(* PLC project Sem nome, Desconhecido Sem nome 1 *)
(* stored: creationDateTime 2019-12-04T19:50:12, modificationDateTime 2019-12-09T14:24:14 *)

PROGRAM Teste1
  VAR
    LIGA_PID AT %QX0.0 : BOOL;
    AUTO_PID AT %QX0.1 : BOOL;
  END_VAR
  VAR RETAIN
    SP AT %MD0 : REAL;
  END_VAR
  VAR
    VP AT %MD1 : REAL;
    SC AT %MD2 : REAL;
  END_VAR
  VAR RETAIN
    KP AT %MD3 : REAL;
    TI AT %MD4 : REAL;
    TD AT %MD5 : REAL;
  END_VAR
  VAR
    VP_RAW AT %IW100 : UINT;
    SC_RAW AT %QW101 : UINT;
  END_VAR
  VAR
    PID0 : PID;
  END_VAR

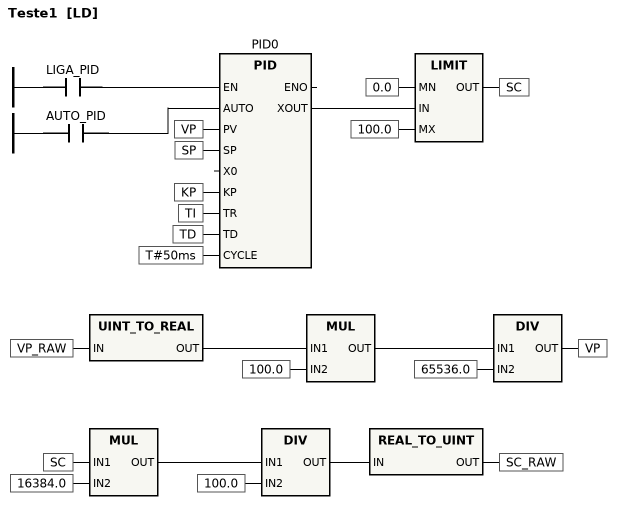
(* LD diagram, written out as Structured Text *)
VP := UINT_TO_REAL(VP_RAW) * 100.0 / 65536.0;
PID0(EN := LIGA_PID, AUTO := AUTO_PID, PV := VP, SP := SP, KP := KP, TR := TI, TD := TD, CYCLE := T#50ms);
SC := LIMIT(0.0, PID0.XOUT, 100.0);
SC_RAW := REAL_TO_UINT(SC * 16384.0 / 100.0);
END_PROGRAM

CONFIGURATION Config0
  RESOURCE Res0 ON PLC
    TASK task0(INTERVAL := T#50ms, PRIORITY := 0);
    PROGRAM instance0 WITH task0 : Teste1;
  END_RESOURCE
END_CONFIGURATION
